Staubli VAL3: start.pgx

program start()
begin

  clearBuffer(soTcpClient)
  movej(jHome,tGreiferM,mUsedSpeed)
  open(tGreiferM)
  open(tGreiferS)


  taskCreate "TCP-Server", 10, TCPserver()

  taskCreate "p&p", 5, PickPlace()

  taskCreate "Vereinzeln", 5, Vereinzeln()



  movej(jHome,tGreiferM,mUsedSpeed)
  waitEndMove()

end
